// Mitsubishi GX Works2 project: Operações_estruturada_02.10   PLC: Q03UDV

// task Task_01 (event TRUE, interval 0, priority 31): POU_01

PROGRAM POU_01
VAR
  CTD_1 : CTD;
  CTU_1 : CTU;
END_VAR
(* structured ladder/FBD written out as ST: instructions are called as NAME(EN, inputs, outputs); _pN, _eN, _tN stand for wires *)
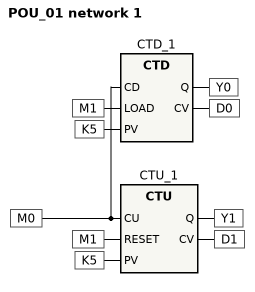
(* network 1 *)
CTD_1(CD := M0, LOAD := M1, PV := K5, Q => Y0, CV => D0);
CTU_1(CU := M0, RESET := M1, PV := K5, Q => Y1, CV => D1);
END_PROGRAM
